PROGRAM Tratadora
VAR
	//Ventilador en tratadora
	TR_S_VE1: Equipo_Motor_No_Rev;
	//
	Eq_TR_sinFalla:BOOL;

	// puerta descarga semilla procesada
	TR_S_V1: Equipo_Valvula_5_2;	//Porta de descarga
	TR_S_V1_CmdAuto:BOOL;	//Comando automático da porta de descarga
	Tmr_PuertaDescarga	:TOF;
	
	fbHomogenizador :Equipo_Motor_ATV320;//Homogenizador
	fbAspersor :Equipo_Motor_ATV320;//Aspersor
	//provisorio
	bHSTR	:BOOL;
	Fin_Dosificado :BOOL;
	
	bHSVE	:BOOL;
	
	Aux_VE:BOOL;
	AbrirDescarga :BOOL;
	
	Tmr_Homogenizado: TON;
	Tiempo_seg_to_TIME_THomog: Tiempo_seg_to_TIME;
	AuxSetTmrPuertaDescarga :TIME;
	AuxSetTmrHomogenizado	:TIME;
	DetenerHomogenizador: BOOL;
	MarchaAutoAspersor: BOOL;
	Dosificar: BOOL;
	PasoDosif: INT;
	VeloAspersorAuto_TR: VeloAspersorAuto;
	TmrDuracionBatch: TON;
	Tiempo_TIME_to_seg_Duracion: Tiempo_TIME_to_seg;
	TBatch:BOOL;
	AuxET_segBatch:DINT;
	CalcPercentual: Percentual;
	TOF_Aspersor: TOF;			//Após a dosagem de produtos, o aspersor fica ligado por 5s 
	TotalizBateladas	:REAL;	//Totalizador dos tempos individuais das bateladas
	TempoBatelada		:REAL; 	//Tempo decorrido da batelada atual
END_VAR
VAR // added by the converter: edge detectors and wires of the graphical bodies
    _w1, _w2, _w3 : BOOL;
    _rt1, _rt2, _rt3 : R_TRIG;
    _ft1 : F_TRIG;
END_VAR

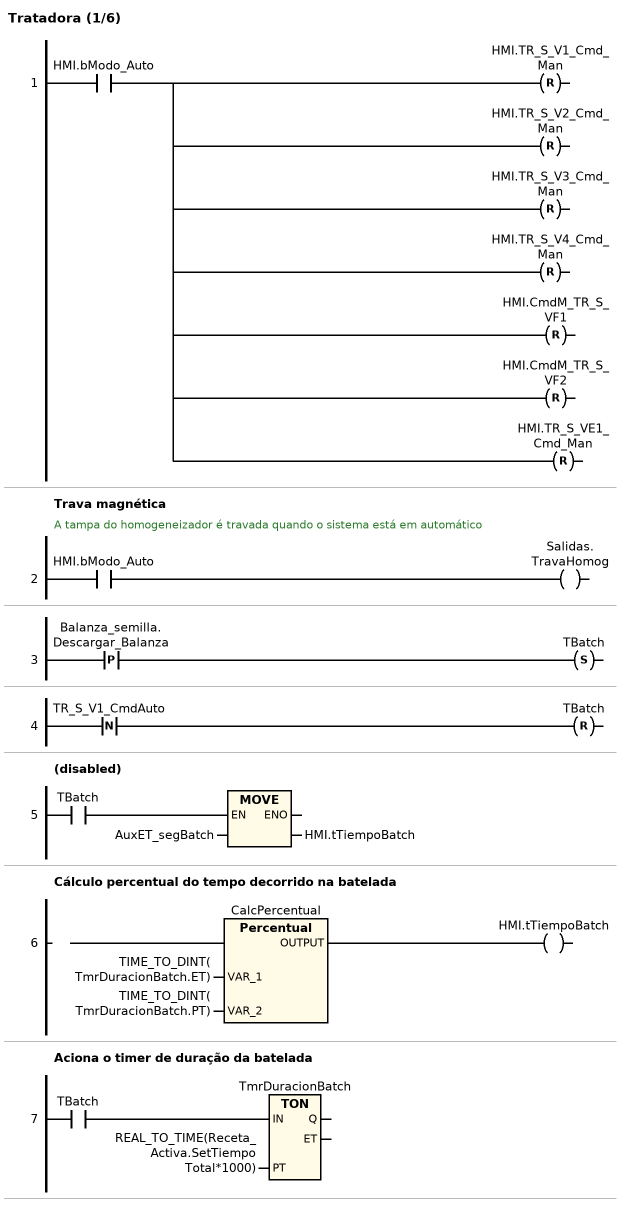
// NETWORK 1
_w1 := HMI.bModo_Auto;
HMI.TR_S_V1_Cmd_Man R= _w1;
HMI.TR_S_V2_Cmd_Man R= _w1;
HMI.TR_S_V3_Cmd_Man R= _w1;
HMI.TR_S_V4_Cmd_Man R= _w1;
HMI.CmdM_TR_S_VF1 R= _w1;
HMI.CmdM_TR_S_VF2 R= _w1;
HMI.TR_S_VE1_Cmd_Man R= _w1;

// NETWORK 2: Trava magnética
// A tampa do homogeneizador é travada quando o sistema está em automático
Salidas.TravaHomog := HMI.bModo_Auto;

// NETWORK 3
_rt1(CLK := Balanza_semilla.Descargar_Balanza);
TBatch S= _rt1.Q;

// NETWORK 4
_ft1(CLK := TR_S_V1_CmdAuto);
TBatch R= _ft1.Q;

// NETWORK 5 (disabled)
// IF TBatch THEN HMI.tTiempoBatch := AuxET_segBatch; END_IF

// NETWORK 6: Cálculo percentual do tempo decorrido na batelada
CalcPercentual(VAR_1 := TIME_TO_DINT(TmrDuracionBatch.ET), VAR_2 := TIME_TO_DINT(TmrDuracionBatch.PT)); // Percentual
HMI.tTiempoBatch := CalcPercentual.OUTPUT;

// NETWORK 7: Aciona o timer de duração da batelada
TmrDuracionBatch(IN := TBatch, PT := REAL_TO_TIME(Receta_Activa.SetTiempoTotal*1000)); // TON

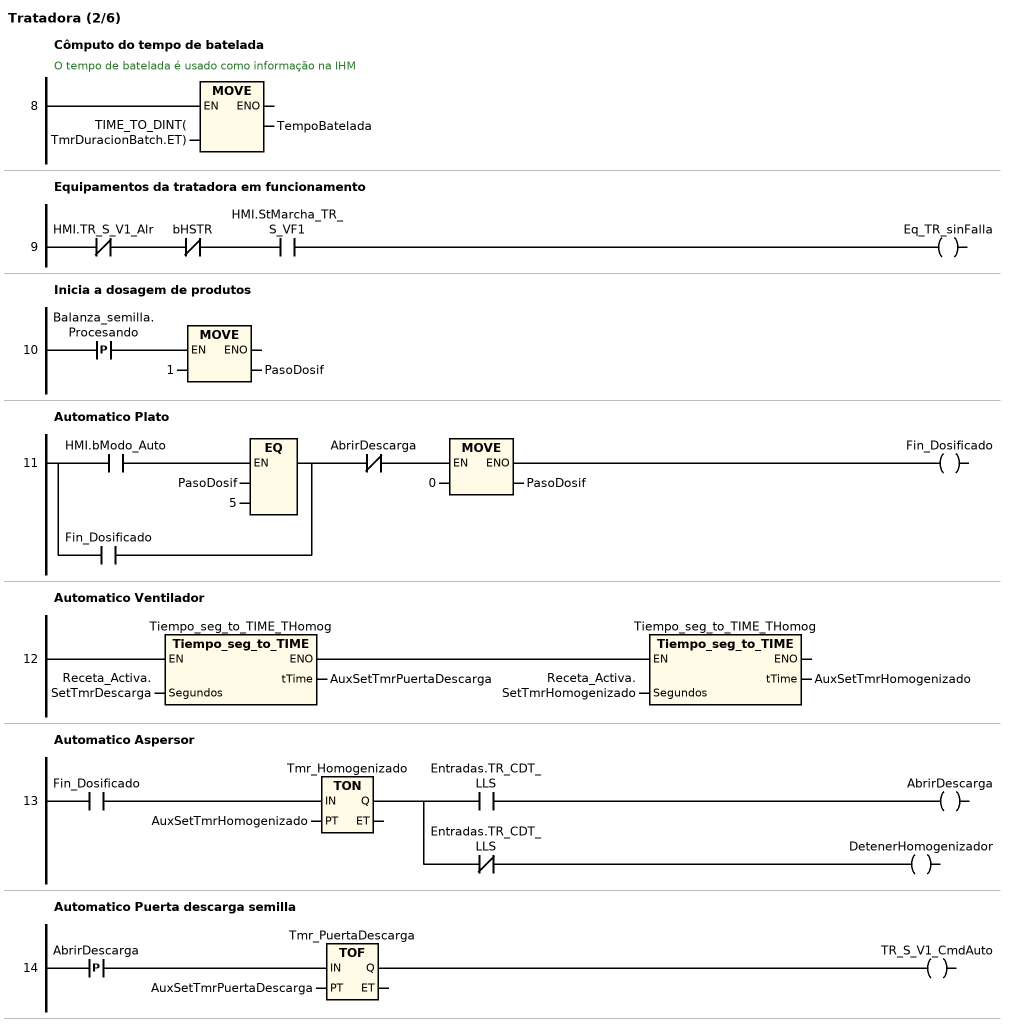
// NETWORK 8: Cômputo do tempo de batelada
// O tempo de batelada é usado como informação na IHM
TempoBatelada := TIME_TO_DINT(TmrDuracionBatch.ET);

// NETWORK 9: Equipamentos da tratadora em funcionamento
Eq_TR_sinFalla := NOT HMI.TR_S_V1_Alr AND NOT bHSTR AND HMI.StMarcha_TR_S_VF1;

// NETWORK 10: Inicia a dosagem de produtos
_rt2(CLK := Balanza_semilla.Procesando);
IF _rt2.Q THEN PasoDosif := 1; END_IF

// NETWORK 11: Automatico Plato
_w2 := (HMI.bModo_Auto AND PasoDosif = 5 OR Fin_Dosificado) AND NOT AbrirDescarga;
IF _w2 THEN PasoDosif := 0; END_IF
Fin_Dosificado := _w2;

// NETWORK 12: Automatico Ventilador
Tiempo_seg_to_TIME_THomog(Segundos := Receta_Activa.SetTmrDescarga, tTime => AuxSetTmrPuertaDescarga); // Tiempo_seg_to_TIME
Tiempo_seg_to_TIME_THomog(Segundos := Receta_Activa.SetTmrHomogenizado, tTime => AuxSetTmrHomogenizado); // Tiempo_seg_to_TIME

// NETWORK 13: Automatico Aspersor
Tmr_Homogenizado(IN := Fin_Dosificado, PT := AuxSetTmrHomogenizado); // TON
AbrirDescarga := Tmr_Homogenizado.Q AND Entradas.TR_CDT_LLS;
DetenerHomogenizador := Tmr_Homogenizado.Q AND NOT Entradas.TR_CDT_LLS;

// NETWORK 14: Automatico Puerta descarga semilla
_rt3(CLK := AbrirDescarga);
Tmr_PuertaDescarga(IN := _rt3.Q, PT := AuxSetTmrPuertaDescarga); // TOF
TR_S_V1_CmdAuto := Tmr_PuertaDescarga.Q;

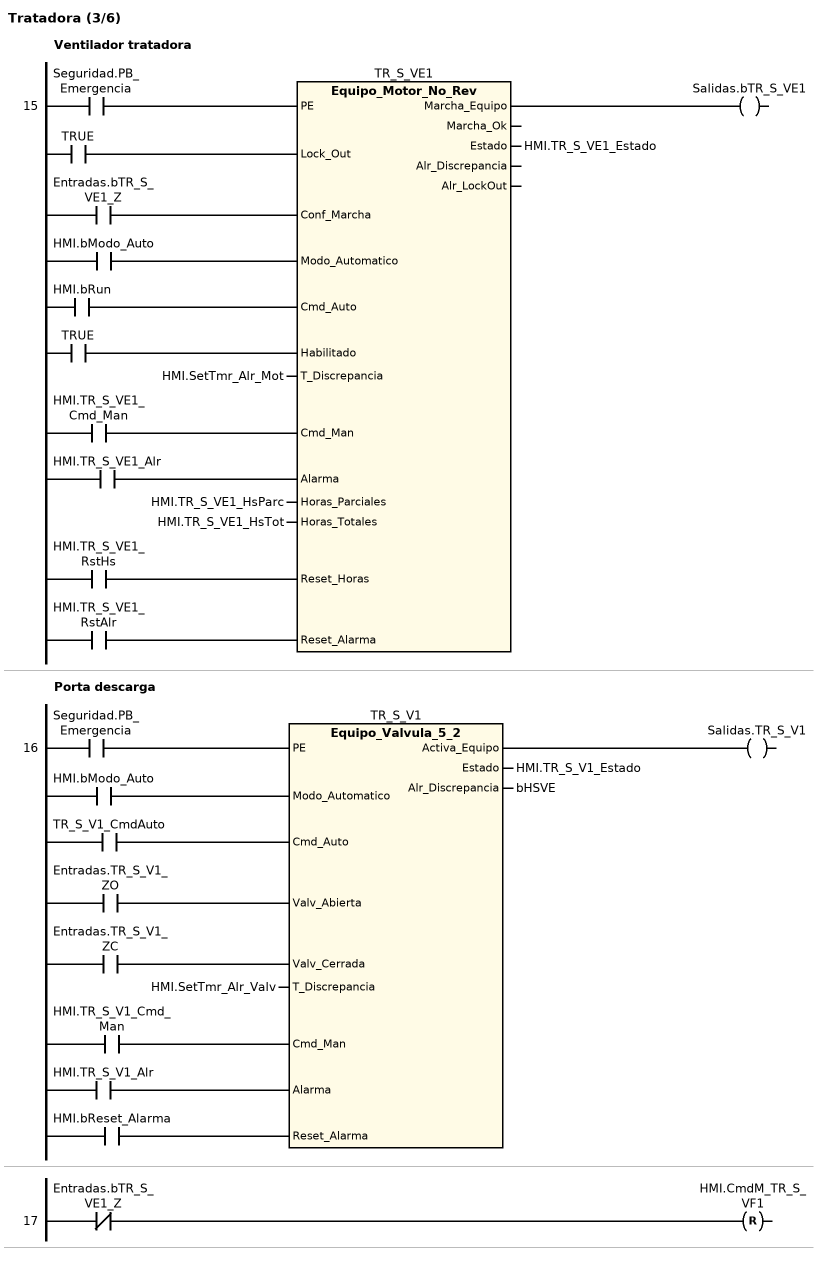
// NETWORK 15: Ventilador tratadora
TR_S_VE1(
    PE := Seguridad.PB_Emergencia,
    Lock_Out := TRUE,
    Conf_Marcha := Entradas.bTR_S_VE1_Z,
    Modo_Automatico := HMI.bModo_Auto,
    Cmd_Auto := HMI.bRun,
    Habilitado := TRUE,
    T_Discrepancia := HMI.SetTmr_Alr_Mot,
    Cmd_Man := HMI.TR_S_VE1_Cmd_Man,
    Alarma := HMI.TR_S_VE1_Alr,
    Horas_Parciales := HMI.TR_S_VE1_HsParc,
    Horas_Totales := HMI.TR_S_VE1_HsTot,
    Reset_Horas := HMI.TR_S_VE1_RstHs,
    Reset_Alarma := HMI.TR_S_VE1_RstAlr,
    Estado => HMI.TR_S_VE1_Estado); // Equipo_Motor_No_Rev
Salidas.bTR_S_VE1 := TR_S_VE1.Marcha_Equipo;

// NETWORK 16: Porta descarga
TR_S_V1(
    PE := Seguridad.PB_Emergencia,
    Modo_Automatico := HMI.bModo_Auto,
    Cmd_Auto := TR_S_V1_CmdAuto,
    Valv_Abierta := Entradas.TR_S_V1_ZO,
    Valv_Cerrada := Entradas.TR_S_V1_ZC,
    T_Discrepancia := HMI.SetTmr_Alr_Valv,
    Cmd_Man := HMI.TR_S_V1_Cmd_Man,
    Alarma := HMI.TR_S_V1_Alr,
    Reset_Alarma := HMI.bReset_Alarma,
    Estado => HMI.TR_S_V1_Estado,
    Alr_Discrepancia => bHSVE); // Equipo_Valvula_5_2
Salidas.TR_S_V1 := TR_S_V1.Activa_Equipo;

// NETWORK 17
HMI.CmdM_TR_S_VF1 R= NOT Entradas.bTR_S_VE1_Z;

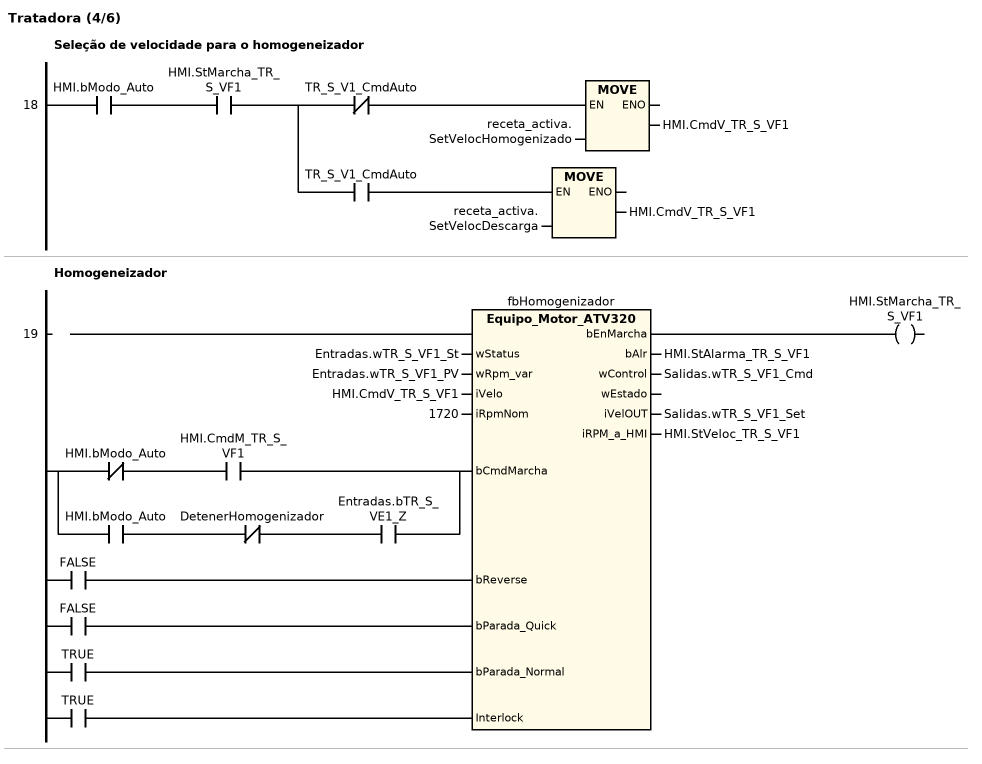
// NETWORK 18: Seleção de velocidade para o homogeneizador
_w3 := HMI.bModo_Auto AND HMI.StMarcha_TR_S_VF1;
IF _w3 AND NOT TR_S_V1_CmdAuto THEN HMI.CmdV_TR_S_VF1 := receta_activa.SetVelocHomogenizado; END_IF
IF _w3 AND TR_S_V1_CmdAuto THEN HMI.CmdV_TR_S_VF1 := receta_activa.SetVelocDescarga; END_IF

// NETWORK 19: Homogeneizador
fbHomogenizador(
    wStatus := Entradas.wTR_S_VF1_St,
    wRpm_var := Entradas.wTR_S_VF1_PV,
    iVelo := HMI.CmdV_TR_S_VF1,
    iRpmNom := 1720,
    bCmdMarcha := NOT HMI.bModo_Auto AND HMI.CmdM_TR_S_VF1 OR HMI.bModo_Auto AND NOT DetenerHomogenizador AND Entradas.bTR_S_VE1_Z,
    bReverse := FALSE,
    bParada_Quick := FALSE,
    bParada_Normal := TRUE,
    Interlock := TRUE,
    bAlr => HMI.StAlarma_TR_S_VF1,
    wControl => Salidas.wTR_S_VF1_Cmd,
    iVelOUT => Salidas.wTR_S_VF1_Set,
    iRPM_a_HMI => HMI.StVeloc_TR_S_VF1); // Equipo_Motor_ATV320
HMI.StMarcha_TR_S_VF1 := fbHomogenizador.bEnMarcha;

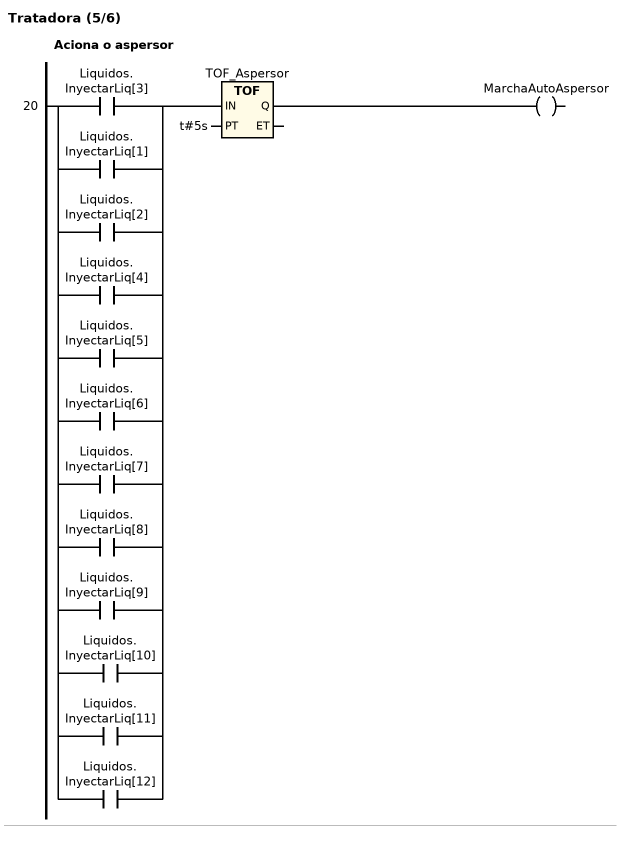
// NETWORK 20: Aciona o aspersor
TOF_Aspersor(IN := Liquidos.InyectarLiq[3] OR Liquidos.InyectarLiq[1] OR Liquidos.InyectarLiq[2] OR Liquidos.InyectarLiq[4] OR Liquidos.InyectarLiq[5] OR Liquidos.InyectarLiq[6] OR Liquidos.InyectarLiq[7] OR Liquidos.InyectarLiq[8] OR Liquidos.InyectarLiq[9] OR Liquidos.InyectarLiq[10] OR Liquidos.InyectarLiq[11] OR Liquidos.InyectarLiq[12], PT := t#5s); // TOF
MarchaAutoAspersor := TOF_Aspersor.Q;

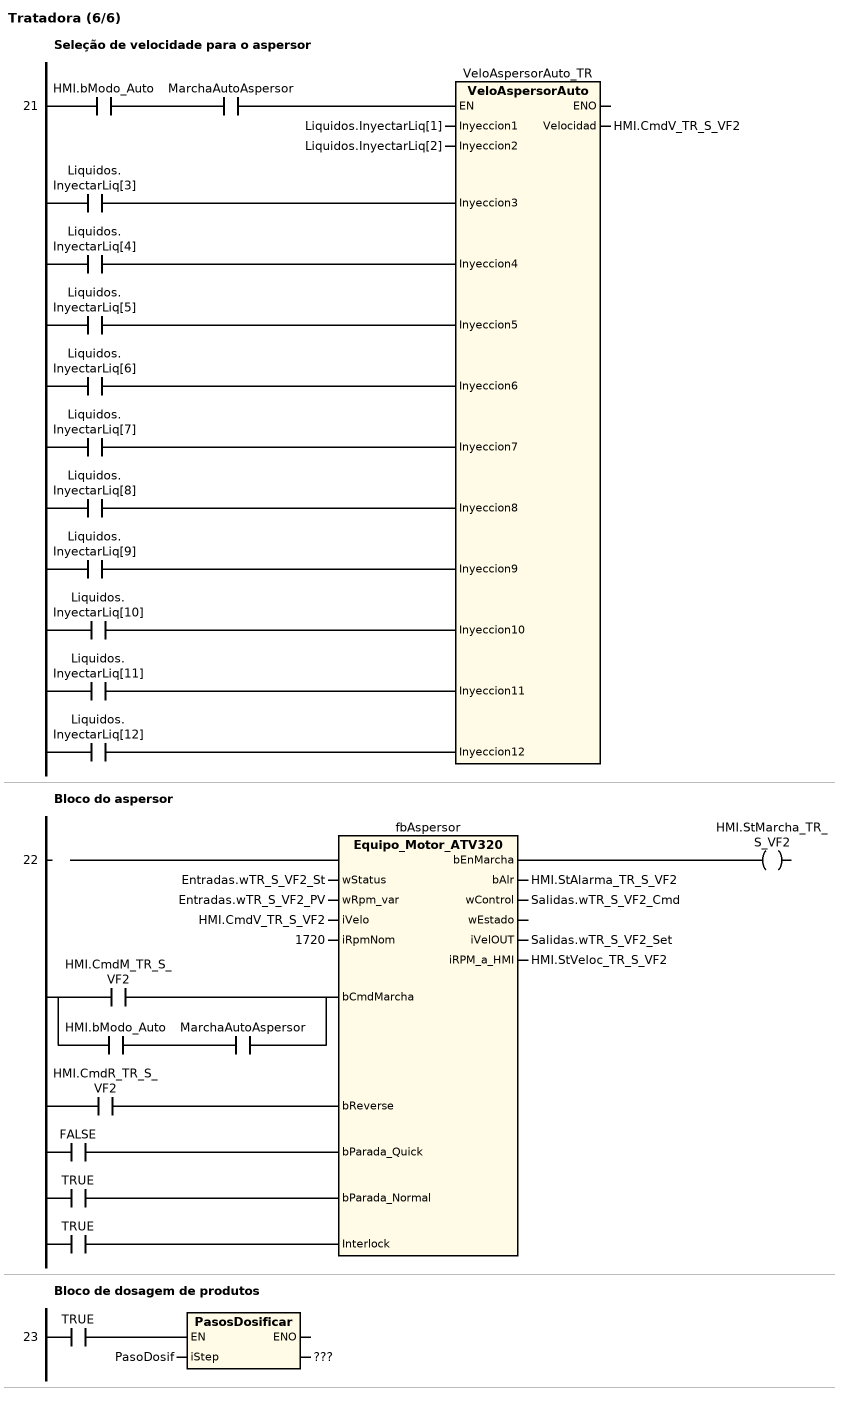
// NETWORK 21: Seleção de velocidade para o aspersor
IF HMI.bModo_Auto AND MarchaAutoAspersor THEN
    VeloAspersorAuto_TR(
        Inyeccion1 := Liquidos.InyectarLiq[1],
        Inyeccion2 := Liquidos.InyectarLiq[2],
        Inyeccion3 := Liquidos.InyectarLiq[3],
        Inyeccion4 := Liquidos.InyectarLiq[4],
        Inyeccion5 := Liquidos.InyectarLiq[5],
        Inyeccion6 := Liquidos.InyectarLiq[6],
        Inyeccion7 := Liquidos.InyectarLiq[7],
        Inyeccion8 := Liquidos.InyectarLiq[8],
        Inyeccion9 := Liquidos.InyectarLiq[9],
        Inyeccion10 := Liquidos.InyectarLiq[10],
        Inyeccion11 := Liquidos.InyectarLiq[11],
        Inyeccion12 := Liquidos.InyectarLiq[12],
        Velocidad => HMI.CmdV_TR_S_VF2); // VeloAspersorAuto
END_IF

// NETWORK 22: Bloco do aspersor
fbAspersor(
    wStatus := Entradas.wTR_S_VF2_St,
    wRpm_var := Entradas.wTR_S_VF2_PV,
    iVelo := HMI.CmdV_TR_S_VF2,
    iRpmNom := 1720,
    bCmdMarcha := HMI.CmdM_TR_S_VF2 OR HMI.bModo_Auto AND MarchaAutoAspersor,
    bReverse := HMI.CmdR_TR_S_VF2,
    bParada_Quick := FALSE,
    bParada_Normal := TRUE,
    Interlock := TRUE,
    bAlr => HMI.StAlarma_TR_S_VF2,
    wControl => Salidas.wTR_S_VF2_Cmd,
    iVelOUT => Salidas.wTR_S_VF2_Set,
    iRPM_a_HMI => HMI.StVeloc_TR_S_VF2); // Equipo_Motor_ATV320
HMI.StMarcha_TR_S_VF2 := fbAspersor.bEnMarcha;

// NETWORK 23: Bloco de dosagem de produtos
PasosDosificar(iStep := PasoDosif);

END_PROGRAM

(* stored: Version 1.1.0.1, ProductVersion 3.1.4024.14
   POU Tratadora: Id {121d19ea-5b58-4225-829d-d2728b309dfb}, SpecialFunc None *)
